// SIMATIC S7-200 project (STEP 7-Micro/WIN), CPU 224XP REL 02.01

SYMBOL_TABLE 符号表
LuTangWen        VD0      // 炉膛温度
YanQiWenDu       VD4      // 烟气温度
LuTangFuYa       VD8      // 炉膛负压
ChuShuiWenDu     VD12     // 出水温度
LuPaiFanKui      VD16     // 炉排反馈
YangHanLiang     VD56     // 烟气氧含量
GuFengFanKui     VD24     // 鼓风反馈
YinFengFanKui    VD28     // 引凤反馈
ShiWaiWenDu      VD36     // 室外温度
ZhaoDu           VD32     // 室外照度
HuiShuiWenDu     VD40     // 回水温度
炉膛负压1            VD104    // 炉膛负压1
引风频率给定           VD200
引风频率死区           VD204
鼓风频率给定           VD300
鼓风频率死区           VD304
炉排频率给定           VD400
炉排频率死区           VD404
上位停止             M0.1
上位启动             M0.0
引至鼓延时间           MW2
鼓至炉排延时时间         MW4
炉排至鼓风停止时间        MW6
鼓风至引凤停止时间        MW8
END_SYMBOL_TABLE

ORGANIZATION_BLOCK 主程序:OB1
TITLE=这个S7-200 PLC程序是为柳河4站的工业锅炉设计的半自动控制系统，包含主程序OB1和子程序SBR0、SBR2、SBR3，为柳河4站的工业锅炉设计半自动控制系统，通过控制引风机、鼓风机和炉排调节燃烧过程。
// 操作人员通过上位机发送启动信号置位引风机启动，经过设定的延时600个时间单位后触发鼓风机启动，再经过设定的延时300个时间单位后激活炉排启动，逐步建立稳定的燃烧环境。
// 在运行过程中，系统实时采集炉膛温度、烟气温度、出水温度等参数，通过输入模拟量转换处理。同时采集回水温度、室外温度、烟气氧含量和室外照度等参数，通过转换处理后，用于监控和控制锅炉状态。例如，炉膛温度帮助判断燃烧状态，烟气氧含量反映燃烧效率。
// 系统根据引风频率给定与引风反馈的比较结果进行调节，引风频率增加只有在差值大于死区时置位，引风频率减少则在差值小于0且超出死区时激活。此外，鼓风频率调节依赖鼓风频率给定与鼓风反馈的差值，炉排频率调节基于炉排频率给定与炉排反馈的差值，确保运行平稳。
// 当启动信号复位时，首先复位炉排启动，经过设定的延时300个时间单位后复位鼓风机启动，再经过设定的延时300个时间单位后复位引风机启动，保证锅炉逐步冷却并安全停机。
BEGIN
Network 1
LD     SM0.1
MOVD   2, 引风频率死区:VD204
MOVD   2, 鼓风频率死区:VD304
MOVD   2, 炉排频率死区:VD404
MOVW   600, 引至鼓延时间:MW2
MOVW   300, 鼓至炉排延时时间:MW4
MOVW   300, 炉排至鼓风停止时间:MW6
MOVW   300, 鼓风至引凤停止时间:MW8
Network 2
LD     SM0.0
CALL   输入模拟量转换:SBR0
Network 3
LD     I0.0
CALL   控制:SBR2
Network 4
LDN    I0.0
R      Q0.0, 3
Network 5
LD     SM0.0
CALL   炉膛负压百分数转换:SBR3
END_ORGANIZATION_BLOCK

SUBROUTINE_BLOCK 输入模拟量转换:SBR0
TITLE=程序注释
BEGIN
Network 1 // 网络标题
// EXP1
// 
LD     SM0.0
CALL   Scale_I_to_R:SBR1, AIW4, 32000, 6400, 1300.0, 0.0, LuTangWen:VD0
CALL   Scale_I_to_R:SBR1, AIW6, 32000, 6400, 1300.0, 0.0, YanQiWenDu:VD4
CALL   Scale_I_to_R:SBR1, AIW10, 32000, 6400, 100.0, 0.0, ChuShuiWenDu:VD12
Network 2 // 题
// EXP2
// 
LD     SM0.0
CALL   Scale_I_to_R:SBR1, AIW14, 32000, 0, 50.0, 0.0, LuPaiFanKui:VD16
CALL   Scale_I_to_R:SBR1, AIW16, 32000, 0, 50.0, 0.0, GuFengFanKui:VD24
CALL   Scale_I_to_R:SBR1, AIW18, 32000, 0, 50.0, 0.0, YinFengFanKui:VD28
Network 3 // 网络标题
// EXP3
// 
LD     SM0.0
CALL   Scale_I_to_R:SBR1, AIW20, 32000, 6400, 20.6, 0.0, YangHanLiang:VD56
CALL   Scale_I_to_R:SBR1, AIW24, 32000, 6400, 200000.0, 0.0, ZhaoDu:VD32
CALL   Scale_I_to_R:SBR1, AIW22, 32000, 6400, 60.0, -26.0, ShiWaiWenDu:VD36
CALL   Scale_I_to_R:SBR1, AIW26, 32000, 6400, 100.0, 0.0, HuiShuiWenDu:VD40
Network 27 // 网络标题
// 网络注释
END_SUBROUTINE_BLOCK

// SBR1: protected block, not included

SUBROUTINE_BLOCK 控制:SBR2
TITLE=子程序注释
BEGIN
Network 1 // 网络标题
// 引风
LD     Q0.0
MOVR   引风频率给定:VD200, VD212
AENO
-R     YinFengFanKui:VD28, VD212
AENO
LPS
AR>    VD212, 引风频率死区:VD204
=      Q0.5
LPP
AR<    VD212, 0.0
MOVR   0.0, VD208
AENO
-R     引风频率死区:VD204, VD208
AENO
AR<    VD212, VD208
=      Q0.6
Network 2 // 网络标题
// 鼓风
LD     Q0.1
MOVR   鼓风频率给定:VD300, VD312
AENO
-R     GuFengFanKui:VD24, VD312
AENO
LPS
AR>    VD312, 引风频率死区:VD204
=      Q0.3
LPP
AR<    VD312, 0.0
MOVR   0.0, VD308
AENO
-R     鼓风频率死区:VD304, VD308
AENO
AR<    VD312, VD308
=      Q0.4
Network 3 // 网络标题
// 鼓风
LD     Q0.2
MOVR   炉排频率给定:VD400, VD412
AENO
-R     LuPaiFanKui:VD16, VD412
AENO
LPS
AR>    VD412, 炉排频率死区:VD404
=      Q1.0
LPP
AR<    VD412, 0.0
MOVR   0.0, VD408
AENO
-R     炉排频率死区:VD404, VD408
AENO
AR<    VD412, VD408
=      Q1.1
Network 4 // 启动
// 引凤启动
LD     上位启动:M0.0
S      Q0.0, 1
TON    T37, 引至鼓延时间:MW2
Network 5
// 鼓风启动
LD     T37
S      Q0.1, 1
TON    T38, 鼓至炉排延时时间:MW4
Network 6
// 炉排启动
LD     T38
S      Q0.2, 1
Network 8
LDN    上位启动:M0.0
R      T37, 2
R      Q0.2, 1
TON    T39, 炉排至鼓风停止时间:MW6
Network 9
LD     T39
R      Q0.1, 1
TON    T40, 鼓风至引凤停止时间:MW8
Network 10
LD     T40
R      Q0.0, 1
END_SUBROUTINE_BLOCK

SUBROUTINE_BLOCK 炉膛负压百分数转换:SBR3
TITLE=子程序注释
BEGIN
Network 1 // 网络标题
// 网络注释
LD     SM0.0
CALL   Scale_I_to_R:SBR1, AIW8, 32000, 6400, 150.0, -50.0, LuTangFuYa:VD8
Network 2
LD     SM0.0
MOVR   LuTangFuYa:VD8, VD100
AENO
+R     50.0, VD100
AENO
MOVR   VD100, 炉膛负压1:VD104
/R     2.0, 炉膛负压1:VD104
END_SUBROUTINE_BLOCK

// SBR4: protected block, not included
